(* CODESYS project lab_1.project

Project tree, tasks and I/O mapping:
  Device : CODESYS Control Win V3, 3S - Smart Software Solutions GmbH, order no. 305021, version 3.5.5.50
    application Application
      libraries: Standard, * (System)
      task MainTask (cyclic, interval t#20ms, priority 1) calls Task
      task VISU_TASK (cyclic, interval 100 ms, priority 31) calls VisuElems.Visu_Prg
      program Task [ST]
      global variables GVL
      visualisation Visualization
  visualisation Visualization
  text list GlobalTextList
*)

// Device/Application/GVL
VAR_GLOBAL
	TEMPER_IN:REAL := 15;
	OPEN_VAL:REAL := 0;
END_VAR

// Device/Application/Task
PROGRAM Task
VAR
	TEMPER_MIN:REAL := 25;
	TEMPER_MAX:REAL := 35;
	
	OPEN_MIN:INT := 0;
	OPEN_MAX:INT := 10;
	
	PROP:REAL;
END_VAR

IF TEMPER_IN >= TEMPER_MIN AND TEMPER_IN < TEMPER_MAX THEN
	PROP:=(TEMPER_IN-TEMPER_MIN)/(TEMPER_MAX-TEMPER_MIN);
	OPEN_VAL:=REAL_TO_INT(PROP * OPEN_MAX);
ELSIF TEMPER_IN < TEMPER_MIN THEN
	OPEN_VAL:=OPEN_MIN;
ELSE
	OPEN_VAL:=OPEN_MAX;
END_IF

END_PROGRAM

// /Visualization
VISUALIZATION Visualization  // 2x2
END_VISUALIZATION

// Device/Application/Visualization
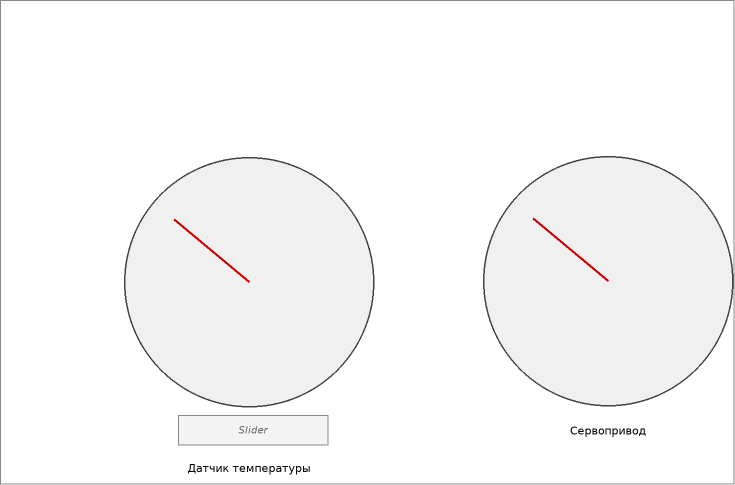
VISUALIZATION Visualization  // 735x485
    Slider (178,415 150x30), variable: TEMPER_IN, scale 15..40
    Label (174,454 150x29), "Датчик температуры"
    Meter360 (483,156 250x250), value: OPEN_VAL, style: Meter-Meter360-Blue, scale format: %.1f, scale 0..10
    Label (533,416 150x30), "Сервопривод"
    Meter360 (124,157 250x250), value: TEMPER_IN, style: Meter-Meter360-Green, scale format: %.1f, scale 15..40
END_VISUALIZATION
